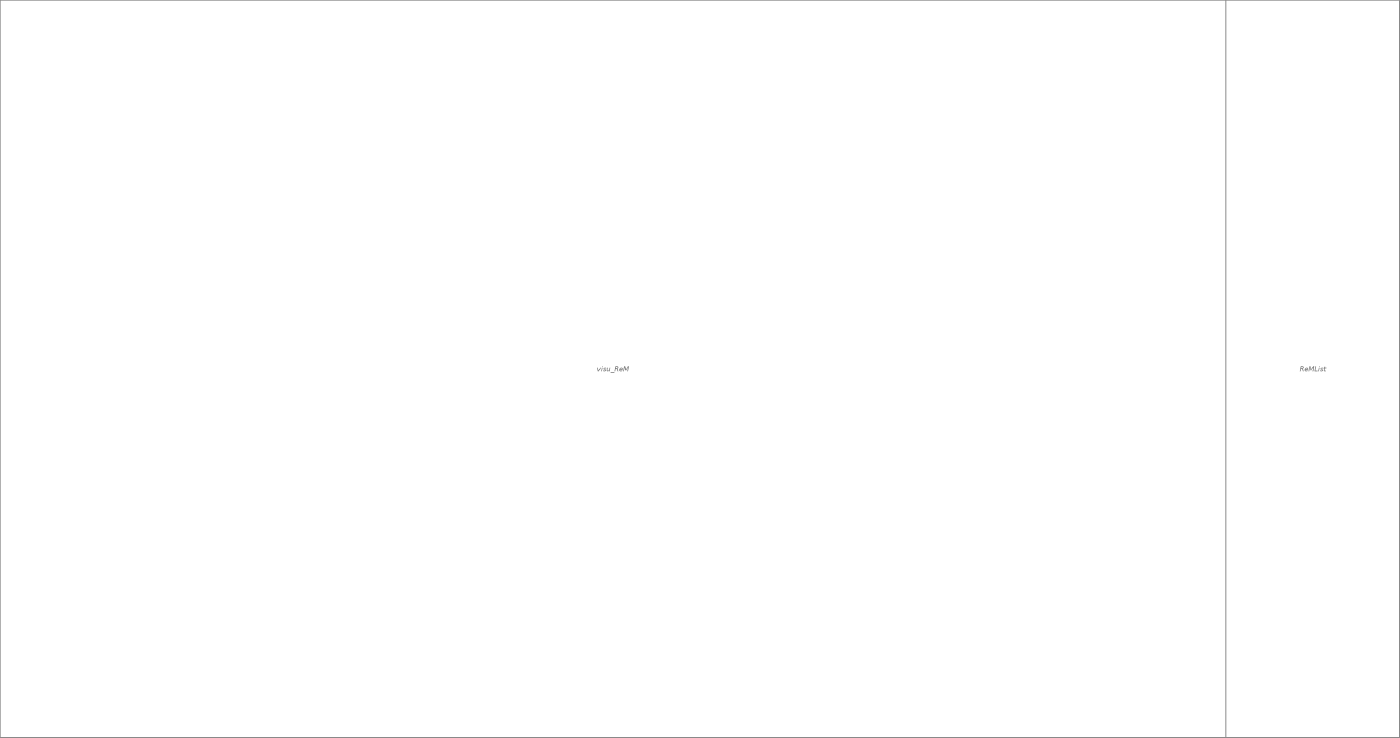
VISUALIZATION visu_main  // 2048x1080
    TabControl (1793,0 255x1080)
        shows ReMList()
        shows PMList()
        shows OtherList()
        shows Visualization_4()
        [0]: TabTitle=ReM
        [2]: TabTitle=Others
    Frame (0,0 1793x1080), frame switch variable: G_HMI.iMainFrame
        shows visu_ReM()
        shows visu_PM()
END_VISUALIZATION

(* stored: Version 1.1.0.1, ProductVersion 3.1.4024.12
   Visu visu_main: Id {27f18664-69ba-41bf-9a81-29f5cd36101a} *)
